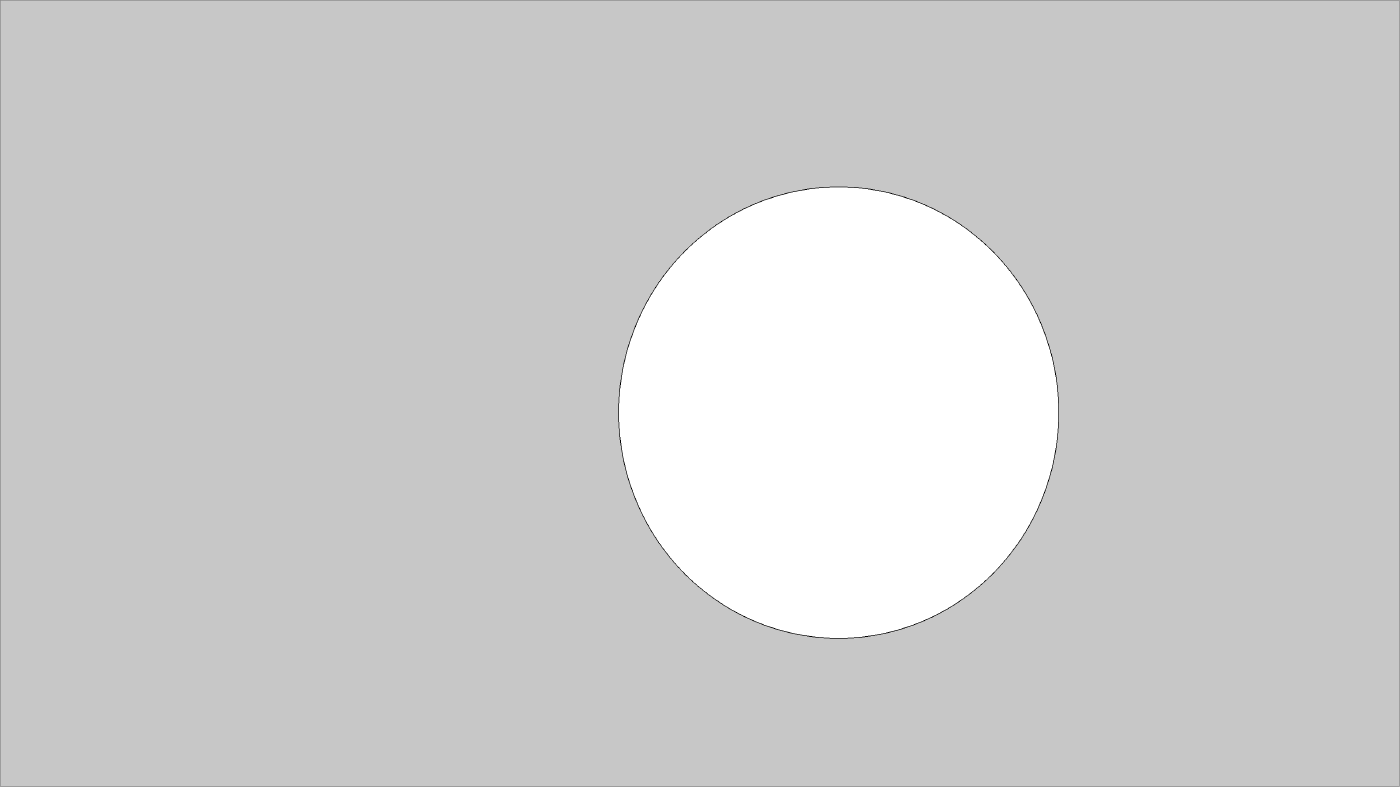
VISUALIZATION Home  // 1920x1080
    Ellipse (848,256 604x620)
        OnMouseClick: change screen: DiagnosticoFB
END_VISUALIZATION

(* stored: Version 1.1.0.1, ProductVersion 3.1.4024.12
   Visu Home: Id {f7a066aa-51fa-41a5-a125-f7a911912ae5} *)
